// TIA Portal V19 export
FUNCTION "FC902_SafetyLogic" : Void   // FC902, F_LAD
{ S7_Optimized_Access := 'TRUE' }
// stored: AutoNumber false
BEGIN

REGION Network 1: Global Emergency Stop Cell
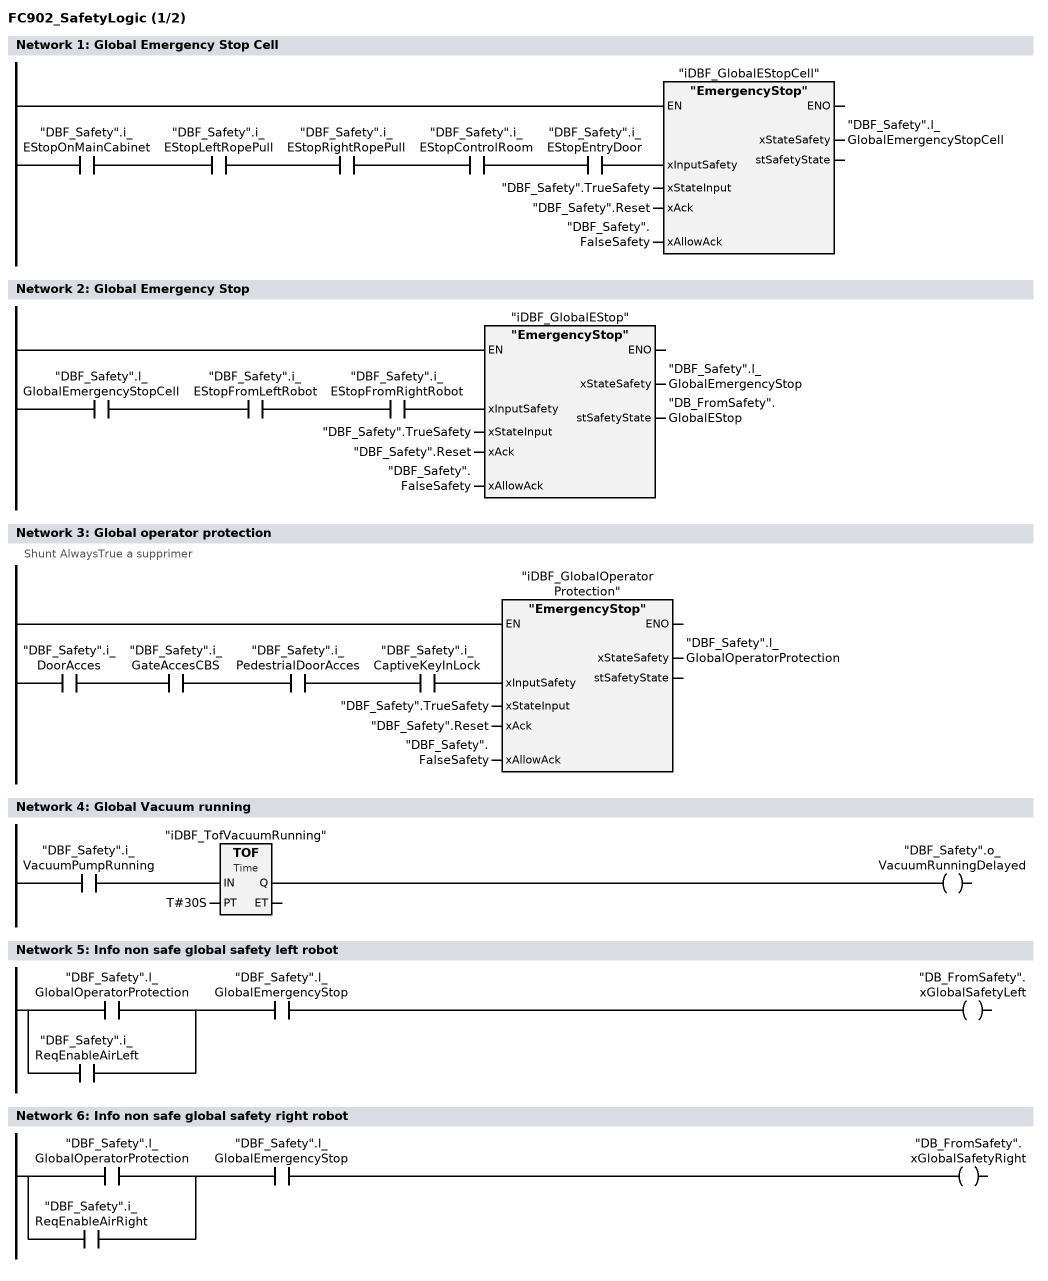
   RUNG wire#powerrail
      "iDBF_GlobalEStopCell"(xInputSafety := wire#w1, xStateInput := "DBF_Safety".TrueSafety, xAck := "DBF_Safety".Reset, xAllowAck := "DBF_Safety".FalseSafety, xStateSafety => "DBF_Safety".l_GlobalEmergencyStopCell, stSafetyState =>)
   END_RUNG
   RUNG wire#powerrail
      Contact( "DBF_Safety".i_EStopOnMainCabinet )
      Contact( "DBF_Safety".i_EStopLeftRopePull )
      Contact( "DBF_Safety".i_EStopRightRopePull )
      Contact( "DBF_Safety".i_EStopControlRoom )
      Contact( "DBF_Safety".i_EStopEntryDoor )
   END_RUNG wire#w1
   // the same network as SCL:
   "iDBF_GlobalEStopCell"(xInputSafety := "DBF_Safety".i_EStopOnMainCabinet AND "DBF_Safety".i_EStopLeftRopePull AND "DBF_Safety".i_EStopRightRopePull AND "DBF_Safety".i_EStopControlRoom AND "DBF_Safety".i_EStopEntryDoor,   // "EmergencyStop"
                          xStateInput := "DBF_Safety".TrueSafety,
                          xAck := "DBF_Safety".Reset,
                          xAllowAck := "DBF_Safety".FalseSafety,
                          xStateSafety => "DBF_Safety".l_GlobalEmergencyStopCell);
END_REGION

REGION Network 2: Global Emergency Stop
   RUNG wire#powerrail
      "iDBF_GlobalEStop"(xInputSafety := wire#w1, xStateInput := "DBF_Safety".TrueSafety, xAck := "DBF_Safety".Reset, xAllowAck := "DBF_Safety".FalseSafety, xStateSafety => "DBF_Safety".l_GlobalEmergencyStop, stSafetyState => "DB_FromSafety".GlobalEStop)
   END_RUNG
   RUNG wire#powerrail
      Contact( "DBF_Safety".l_GlobalEmergencyStopCell )
      Contact( "DBF_Safety".i_EStopFromLeftRobot )
      Contact( "DBF_Safety".i_EStopFromRightRobot )
   END_RUNG wire#w1
   // the same network as SCL:
   "iDBF_GlobalEStop"(xInputSafety := "DBF_Safety".l_GlobalEmergencyStopCell AND "DBF_Safety".i_EStopFromLeftRobot AND "DBF_Safety".i_EStopFromRightRobot,   // "EmergencyStop"
                      xStateInput := "DBF_Safety".TrueSafety,
                      xAck := "DBF_Safety".Reset,
                      xAllowAck := "DBF_Safety".FalseSafety,
                      xStateSafety => "DBF_Safety".l_GlobalEmergencyStop,
                      stSafetyState => "DB_FromSafety".GlobalEStop);
END_REGION

REGION Network 3: Global operator protection
   // Shunt AlwaysTrue a supprimer
   RUNG wire#powerrail
      "iDBF_GlobalOperatorProtection"(xInputSafety := wire#w1, xStateInput := "DBF_Safety".TrueSafety, xAck := "DBF_Safety".Reset, xAllowAck := "DBF_Safety".FalseSafety, xStateSafety => "DBF_Safety".l_GlobalOperatorProtection, stSafetyState =>)
   END_RUNG
   RUNG wire#powerrail
      Contact( "DBF_Safety".i_DoorAcces )
      Contact( "DBF_Safety".i_GateAccesCBS )
      Contact( "DBF_Safety".i_PedestrialDoorAcces )
      Contact( "DBF_Safety".i_CaptiveKeyInLock )
   END_RUNG wire#w1
   // the same network as SCL:
   "iDBF_GlobalOperatorProtection"(xInputSafety := "DBF_Safety".i_DoorAcces AND "DBF_Safety".i_GateAccesCBS AND "DBF_Safety".i_PedestrialDoorAcces AND "DBF_Safety".i_CaptiveKeyInLock,   // "EmergencyStop"
                           xStateInput := "DBF_Safety".TrueSafety,
                           xAck := "DBF_Safety".Reset,
                           xAllowAck := "DBF_Safety".FalseSafety,
                           xStateSafety => "DBF_Safety".l_GlobalOperatorProtection);
END_REGION

REGION Network 4: Global Vacuum running
   RUNG wire#powerrail
      Contact( "DBF_Safety".i_VacuumPumpRunning )
      { S7_Templates := "[time_type := Time, codedbool_type := DInt]" } "iDBF_TofVacuumRunning".TOF(pt := T#30S, et =>)
      Coil( "DBF_Safety".o_VacuumRunningDelayed )
   END_RUNG
   // the same network as SCL:
   "iDBF_TofVacuumRunning".TOF(IN := "DBF_Safety".i_VacuumPumpRunning, PT := T#30S);
   "DBF_Safety".o_VacuumRunningDelayed := "iDBF_TofVacuumRunning".Q;
END_REGION

REGION Network 5: Info non safe global safety left robot
   RUNG wire#powerrail
      Contact( "DBF_Safety".l_GlobalOperatorProtection )
      wire#w1
      Contact( "DBF_Safety".l_GlobalEmergencyStop )
      Coil( "DB_FromSafety".xGlobalSafetyLeft )
   END_RUNG
   RUNG wire#powerrail
      Contact( "DBF_Safety".i_ReqEnableAirLeft )
   END_RUNG wire#w1
   // the same network as SCL:
   "DB_FromSafety".xGlobalSafetyLeft := ("DBF_Safety".l_GlobalOperatorProtection OR "DBF_Safety".i_ReqEnableAirLeft) AND "DBF_Safety".l_GlobalEmergencyStop;
END_REGION

REGION Network 6: Info non safe global safety right robot
   RUNG wire#powerrail
      Contact( "DBF_Safety".l_GlobalOperatorProtection )
      wire#w1
      Contact( "DBF_Safety".l_GlobalEmergencyStop )
      Coil( "DB_FromSafety".xGlobalSafetyRight )
   END_RUNG
   RUNG wire#powerrail
      Contact( "DBF_Safety".i_ReqEnableAirRight )
   END_RUNG wire#w1
   // the same network as SCL:
   "DB_FromSafety".xGlobalSafetyRight := ("DBF_Safety".l_GlobalOperatorProtection OR "DBF_Safety".i_ReqEnableAirRight) AND "DBF_Safety".l_GlobalEmergencyStop;
END_REGION

REGION Network 7: Enable air pressure supply for left robot
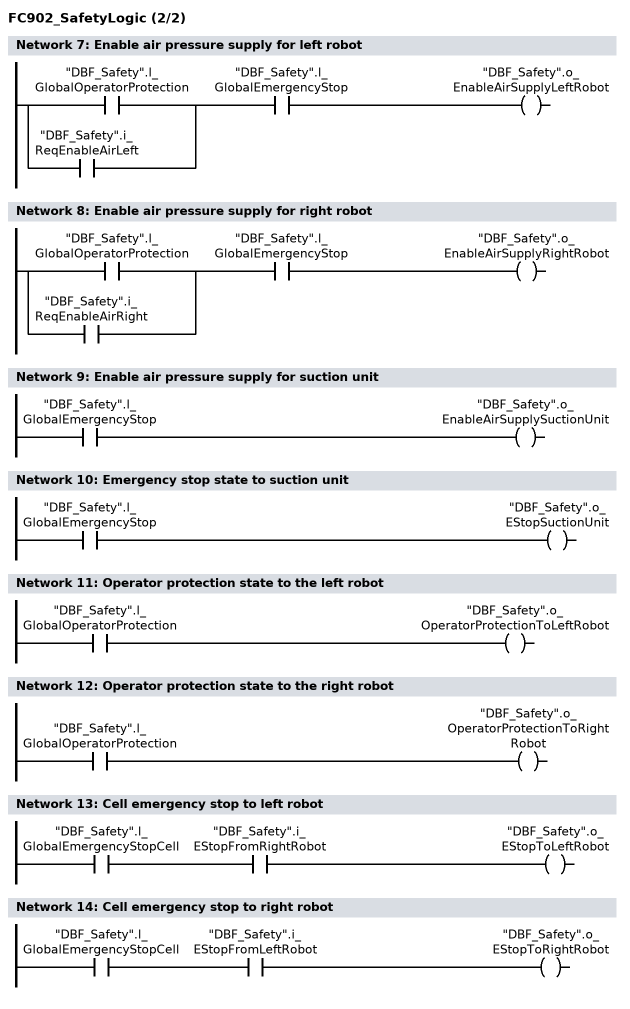
   RUNG wire#powerrail
      Contact( "DBF_Safety".l_GlobalOperatorProtection )
      wire#w1
      Contact( "DBF_Safety".l_GlobalEmergencyStop )
      Coil( "DBF_Safety".o_EnableAirSupplyLeftRobot )
   END_RUNG
   RUNG wire#powerrail
      Contact( "DBF_Safety".i_ReqEnableAirLeft )
   END_RUNG wire#w1
   // the same network as SCL:
   "DBF_Safety".o_EnableAirSupplyLeftRobot := ("DBF_Safety".l_GlobalOperatorProtection OR "DBF_Safety".i_ReqEnableAirLeft) AND "DBF_Safety".l_GlobalEmergencyStop;
END_REGION

REGION Network 8: Enable air pressure supply for right robot
   RUNG wire#powerrail
      Contact( "DBF_Safety".l_GlobalOperatorProtection )
      wire#w1
      Contact( "DBF_Safety".l_GlobalEmergencyStop )
      Coil( "DBF_Safety".o_EnableAirSupplyRightRobot )
   END_RUNG
   RUNG wire#powerrail
      Contact( "DBF_Safety".i_ReqEnableAirRight )
   END_RUNG wire#w1
   // the same network as SCL:
   "DBF_Safety".o_EnableAirSupplyRightRobot := ("DBF_Safety".l_GlobalOperatorProtection OR "DBF_Safety".i_ReqEnableAirRight) AND "DBF_Safety".l_GlobalEmergencyStop;
END_REGION

REGION Network 9: Enable air pressure supply for suction unit
   RUNG wire#powerrail
      Contact( "DBF_Safety".l_GlobalEmergencyStop )
      Coil( "DBF_Safety".o_EnableAirSupplySuctionUnit )
   END_RUNG
   // the same network as SCL:
   "DBF_Safety".o_EnableAirSupplySuctionUnit := "DBF_Safety".l_GlobalEmergencyStop;
END_REGION

REGION Network 10: Emergency stop state to suction unit
   RUNG wire#powerrail
      Contact( "DBF_Safety".l_GlobalEmergencyStop )
      Coil( "DBF_Safety".o_EStopSuctionUnit )
   END_RUNG
   // the same network as SCL:
   "DBF_Safety".o_EStopSuctionUnit := "DBF_Safety".l_GlobalEmergencyStop;
END_REGION

REGION Network 11: Operator protection state to the left robot
   RUNG wire#powerrail
      Contact( "DBF_Safety".l_GlobalOperatorProtection )
      Coil( "DBF_Safety".o_OperatorProtectionToLeftRobot )
   END_RUNG
   // the same network as SCL:
   "DBF_Safety".o_OperatorProtectionToLeftRobot := "DBF_Safety".l_GlobalOperatorProtection;
END_REGION

REGION Network 12: Operator protection state to the right robot
   RUNG wire#powerrail
      Contact( "DBF_Safety".l_GlobalOperatorProtection )
      Coil( "DBF_Safety".o_OperatorProtectionToRightRobot )
   END_RUNG
   // the same network as SCL:
   "DBF_Safety".o_OperatorProtectionToRightRobot := "DBF_Safety".l_GlobalOperatorProtection;
END_REGION

REGION Network 13: Cell emergency stop to left robot
   RUNG wire#powerrail
      Contact( "DBF_Safety".l_GlobalEmergencyStopCell )
      Contact( "DBF_Safety".i_EStopFromRightRobot )
      Coil( "DBF_Safety".o_EStopToLeftRobot )
   END_RUNG
   // the same network as SCL:
   "DBF_Safety".o_EStopToLeftRobot := "DBF_Safety".l_GlobalEmergencyStopCell AND "DBF_Safety".i_EStopFromRightRobot;
END_REGION

REGION Network 14: Cell emergency stop to right robot
   RUNG wire#powerrail
      Contact( "DBF_Safety".l_GlobalEmergencyStopCell )
      Contact( "DBF_Safety".i_EStopFromLeftRobot )
      Coil( "DBF_Safety".o_EStopToRightRobot )
   END_RUNG
   // the same network as SCL:
   "DBF_Safety".o_EStopToRightRobot := "DBF_Safety".l_GlobalEmergencyStopCell AND "DBF_Safety".i_EStopFromLeftRobot;
END_REGION
END_FUNCTION
